Staubli VAL3: delStrArray.pgx

public program delStrArray(string& x_sStrIn[], num x_nNum)
  local num l_nSize
  local num l_i
begin
  //删除字符串数组
  //x_sStrIn:返回的新数组
  //x_nNum:删除数组个数
  //取整
  x_nNum=roundDown(x_nNum)
  //
  l_nSize=size(x_sStrIn)
  if l_nSize<=1
    x_sStrIn=""
    return
  endIf
  //
  if x_nNum>=l_nSize
    x_nNum=l_nSize-1
    x_sStrIn[0]=""
  endIf
  //

  while x_nNum>=1
    delete(x_sStrIn[size(x_sStrIn)-1])
    x_nNum=x_nNum-1
  endWhile

end
